// Mitsubishi GX Works2 project: MY_PULSE_CODE   PLC: Q03UDV

PROGRAM MAIN
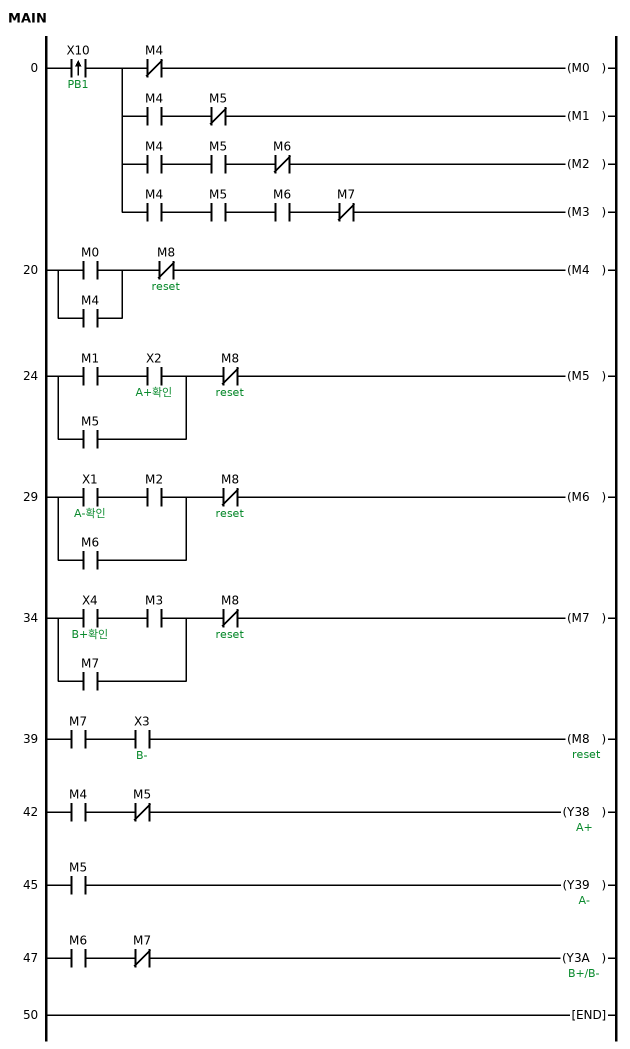
0     LDP     X10  ; PB1
      MPS
      ANI     M4
      OUT     M0
      MRD
      AND     M4
      ANI     M5
      OUT     M1
      MRD
      AND     M4
      AND     M5
      ANI     M6
      OUT     M2
      MPP
      AND     M4
      AND     M5
      AND     M6
      ANI     M7
      OUT     M3
20    LD      M0
      OR      M4
      ANI     M8  ; reset
      OUT     M4
24    LD      M1
      AND     X2  ; A+확인
      OR      M5
      ANI     M8  ; reset
      OUT     M5
29    LD      X1  ; A-확인
      AND     M2
      OR      M6
      ANI     M8  ; reset
      OUT     M6
34    LD      X4  ; B+확인
      AND     M3
      OR      M7
      ANI     M8  ; reset
      OUT     M7
39    LD      M7
      AND     X3  ; B-
      OUT     M8  ; reset
42    LD      M4
      ANI     M5
      OUT     Y38  ; A+
45    LD      M5
      OUT     Y39  ; A-
47    LD      M6
      ANI     M7
      OUT     Y3A  ; B+/B-
50    END
END_PROGRAM
